    // check whether to continue
    if (l_bOk)

      //region @DEBUG
      if (bDebugMode and nDebugLevel==7)
        call printDebug("INFO: state transition ("+toString("",nMotionMode)+" -> "+toString("",l_nNextState)+")",false)
      endIf
      //endregion

      //region @clean_up_motion_task -- if so force motion task to reset motion and/or kill the task
      if (l_bResetMotion)
        // set stop flag (important for velocity mode: reconfiguration without killing task)
        bStopNow=true
      elseIf (l_bKillMotTask)
        // if the current motion task has to be killed, wait until it finishes cleaning up
        bStopNow=true
        wait(bStopNow==false)
        // ... and then kill the task
        taskKill(sMotionTask)
        resetMotion()

        //region @DEBUG
        if (bDebugMode and nDebugLevel==7)
          call printDebug("INFO: motion task killed",false)
        endIf
        //endregion
      endIf
      //endregion

      //region @create_new_motion_task -- create the new motion task if required
      if (l_bKillMotTask)
        switch l_nNextState
          case Staubli:MotionMode.JOINT_TRAJ
            taskCreateSync sMotionTask,nMotionPeriod,bMotionOverrun,motionControl()
          break
          case Staubli:MotionMode.VELOCITY_CTRL
            taskCreateSync sMotionTask,nMotionPeriod,bMotionOverrun,motionCtrlVel()
          break
          default
            l_bOk=false
            //region @DEBUG
            if (bDebugMode and nDebugLevel==7)
              call printDebug("ERROR: unknown next state",false)
            endIf
            //endregion
          break
        endSwitch

        //region @DEBUG
        if (bDebugMode and nDebugLevel==7)
          if (l_bOk)
            call printDebug("INFO: new motion task created",false)
          else
            call printDebug("ERROR: new motion task not created",false)
          endIf
        endIf
        //endregion
      endIf
      //endregion

      // finally update current state if successful
      if (l_bOk)
        if (l_nNextState!=Staubli:MotionMode.INVALID)
          nMotionMode=l_nNextState

          //region @DEBUG
          if (bDebugMode and nDebugLevel==7)
            call printDebug("INFO: set new state ("+toString("",l_nNextState)+")",false)
          endIf
          //endregion
        else
          //region @DEBUG
          if (bDebugMode and nDebugLevel==7)
            call printDebug("WARN: state not set -> invalid ("+toString("",l_nNextState)+")",false)
          endIf
          //endregion
        endIf
      endIf

    endIf

    // sequence task
    delay(0)
  endWhile
end

--- stop.pgx ---
program stop()
begin
  // Copyright (c) 2016, Ocado Technology - Robotics Research Team
  //
  // Licensed under the Apache License, Version 2.0 (the "License");
  // you may not use this file except in compliance with the License.
  // You may obtain a copy of the License at
  //
  //     http://www.apache.org/licenses/LICENSE-2.0
  //
  // Unless required by applicable law or agreed to in writing, software
  // distributed under the License is distributed on an "AS IS" BASIS,
  // WITHOUT WARRANTIES OR CONDITIONS OF ANY KIND, either express or implied.
  // See the License for the specific language governing permissions and
  // limitations under the License.



  resetMotion()
  popUpMsg("Pending movement commands have been cancelled.")

  if nLibLoadError == 0
    call libInterface:clearScreen()
  endIf

  taskKill("streamerTask")
  taskKill("trajPtTask")
  taskKill("motionTask")
  taskKill("screenTask")
  taskKill("htbtTask")

end

--- taskManager.pgx ---
program taskManager()
begin
  // Copyright (c) 2016, Ocado Technology - Robotics Research Team
  //
  // Licensed under the Apache License, Version 2.0 (the "License");
  // you may not use this file except in compliance with the License.
  // You may obtain a copy of the License at
  //
  //     http://www.apache.org/licenses/LICENSE-2.0
  //
  // Unless required by applicable law or agreed to in writing, software
  // distributed under the License is distributed on an "AS IS" BASIS,
  // WITHOUT WARRANTIES OR CONDITIONS OF ANY KIND, either express or implied.
  // See the License for the specific language governing permissions and
  // limitations under the License.

  // taskstatus:
  // -1 : task is not running
  //  0 : stopped
  //  1 : started
  // >1 : VAL3 runtime error

  do

    // create joint state and robot status streamer task to send data to industrial_robot_client
    if taskStatus(sStreamTaskName) == -1
      taskCreateSync sStreamTaskName, nFbkPeriod, bFbkOverrun, dataStreamer()
      wait(taskStatus(sStreamTaskName) != -1)
    endIf

    // create trajectory point task to receive data from industrial_robot_client
    if taskStatus(sTrajPtTaskName) == -1
      taskCreateSync sTrajPtTaskName, nTrajPeriod, bTrajPtOverrun, dataReceiver()
      wait(taskStatus(sTrajPtTaskName) != -1)
    endIf

    // create motion task to synchronously apply motion commands to robot
    if taskStatus(sMotionTaskName) == -1
      taskCreateSync sMotionTaskName, nMotionPeriod, bMotionOverrun, motionControl()
      wait(taskStatus(sMotionTaskName) != -1)
    endIf

    // create asynchronous task to update screen
    if taskStatus(sScreenTaskName) == -1
      taskCreate sScreenTaskName, 10, screenUpdate()
      wait(taskStatus(sScreenTaskName) != -1)
    endIf

    // create asynchronous task to receive heartbeat on port 11002
    if taskStatus(sHtbtTaskName) == -1
      taskCreate sHtbtTaskName, 10, recvHeartbeat()
      wait(taskStatus(sHtbtTaskName) != -1)
    endIf

  until false
end
